// Mitsubishi GX Works2 project: compiler   PLC: FX3G

// global labels: Global1
VAR_GLOBAL
  AM_EVENTS : ARRAY [0..3] OF ST_AM_EVENT;
  AM_ALARMS : ARRAY [0..2] OF ST_AM_ALARM;
END_VAR
VAR_GLOBAL CONSTANT
  c_AM_ALARMS_NUM : INT := 3;
  c_AM_EVENTS_NUM : INT := 3;
END_VAR
VAR_GLOBAL
  MB_CHANNELS : ARRAY [0..2] OF ST_MB_REG_50;
END_VAR
VAR_GLOBAL CONSTANT
  c_MB_CHANNELS_NUM : INT := 2;
END_VAR

// task MAIN (event TRUE, interval 0, priority 31): MAIN
// task AM (event FALSE, interval T#100ms, priority 31): PRG_AM_TEST
// task TCO (event I750, interval 0, priority 26): PRG_TCO_TICKER_50
// task TCO_TEST (event FALSE, interval T#20ms, priority 31): PRG_TEST_TCO_50
// task MB (event FALSE, interval T#20ms, priority 31): PRG_MB_TEST
// user libraries (not included): AlarmManger, Modbus, TimeControl, UtilsV5

PROGRAM MAIN
VAR
  fbHyst : FB_HYST;  (* Heating regulator instance *)
  fbHystCool : FB_HYST_COOL;  (* Cooling regulator instance *)
  fbScaleAI : FB_SCALE_AI;  (* Host PLC analog input scaling instance *)
  fbL02ScaleAI : L02_SCALE_AI;  (* L02 module analog input scaling instance *)
  fbValve3P : FB_VALVE_3P;  (* 3-position valve control instance *)
  xSaveIp : BOOL;  (* Manual trigger: write IP settings (force TRUE) *)
  xValveEnable : BOOL;  (* Manual valve enable input *)
  xIsOnWord : BOOL;  (* F_ISBON result (bit 2 of 16#0004 = TRUE) *)
  xIsOnDword : BOOL;  (* F_DISBON result (bit 2 of 16#00000004 = TRUE) *)
  wSetWord : WORD;  (* F_SETB result (16#0000 with bit 3 set = 16#0008) *)
  dwSetWord : DWORD;  (* F_DSETB result (bit 3 set) *)
  wRstWord : WORD;  (* F_RSTB result (16#000F with bit 2 cleared = 16#000B) *)
  dwRstWord : DWORD;  (* F_DRSTB result (bit 2 cleared) *)
  wSrbWord : WORD;  (* F_SRB result (bit 5 set) *)
  dwSrbWord : DWORD;  (* F_DSRB result (bit 5 set) *)
  iLimit : INT;  (* F_LIMIT result (150 clamped to 100) *)
  iScale : INT;  (* F_SCALE result (50 -> 500) *)
  iScaleNl : INT;  (* F_SCALE_NL result *)
  iIncrement : INT;  (* F_INCN result (2 -> 3) *)
  iShift : INT;  (* F_SHFT result (4 shifted by 2 within 0..5 = 0) *)
  iWorkLeft : INT;  (* F_WORK_LEFT result (25/100 -> 75) *)
  iWorkLeftTime : INT;  (* F_WORK_LEFT_TIME result (25s/100s -> 75) *)
  iValvePos : INT;  (* F_VALVE_POS result (5s/10s -> 500) *)
  rFlt10 : REAL;  (* F_FLT10 result (123 -> 12.3) *)
  xSetIp : BOOL;  (* F_L02_SET_IP result *)
  xMbmov : BOOL;  (* F_MBMOV result *)
  xHystQ : BOOL;  (* FB_HYST output *)
  xHystCoolQ : BOOL;  (* FB_HYST_COOL output *)
  iScaleAIValue : INT;  (* FB_SCALE_AI scaled value *)
  xScaleAIWire : BOOL;  (* FB_SCALE_AI wire error *)
  xScaleAILimit : BOOL;  (* FB_SCALE_AI limit error *)
  xScaleAIMinMax : BOOL;  (* FB_SCALE_AI min/max error *)
  iL02ScaleAIValue : INT;  (* FB_L02_SCALE_AI scaled value *)
  xValveOpen : BOOL;  (* FB_VALVE_3P open command *)
  xValveClose : BOOL;  (* FB_VALVE_3P close command *)
END_VAR
EI(TRUE);

(*
  Utils library smoke test.

  Calls every function ( F_* ) and function block ( FB_* ) OF the Utils library
  with representative test inputs. Results are stored in auto-assigned labels
  so they can be watched in the device monitor.

  Functions exercised:
    F_ISBON / F_DISBON / F_SETB / F_DSETB / F_RSTB / F_DRSTB / F_SRB / F_DSRB
    F_LIMIT / F_SCALE / F_SCALE_NL / F_INCN / F_SHFT
    F_WORK_LEFT / F_WORK_LEFT_TIME / F_VALVE_POS / F_FLT10
    F_L02_SET_IP / F_MBMOV

  Function blocks exercised:
    FB_HYST / FB_HYST_COOL / FB_SCALE_AI / FB_L02_SCALE_AI / FB_VALVE_3P

  Notes:
    - FB_VALVE_3P uses the TCO_DINT_50 ticker AND therefore requires the
      TimeControl library with its TCO timer setup.
    - F_L02_SET_IP, F_MBMOV AND F_SCALE_NL write to R / D devices.
    - Force the xSaveIp / xValveEnable inputs AND watch the result labels.
*)

(* --- Bit check / bit manipulation functions --- *)
xIsOnWord  := F_ISBON(16#0004, 2);
xIsOnDword := F_DISBON(16#00000004, 2);

wSetWord  := F_SETB(16#0000, 3);
dwSetWord := F_DSETB(16#00000000, 3);

wRstWord  := F_RSTB(16#000F, 2);
dwRstWord := F_DRSTB(16#0000000F, 2);

wSrbWord  := F_SRB(16#0000, 5, TRUE);
dwSrbWord := F_DSRB(16#00000000, 5, TRUE);

(* --- Value / index functions --- *)
iLimit     := F_LIMIT(100, 150, 0);
iScale     := F_SCALE(50, 0, 100, 0, 1000);
iScaleNl   := F_SCALE_NL(2, 100, 50);  (* writes D100..D103 *)

iIncrement := F_INCN(TRUE, 2, 5);
iShift     := F_SHFT(2, 4, 5);

(* --- Progress / time functions --- *)
iWorkLeft     := F_WORK_LEFT(25, 100);
iWorkLeftTime := F_WORK_LEFT_TIME(T#25s, T#100s);
iValvePos     := F_VALVE_POS(T#5s, T#10s);

(* --- Filter function (returns REAL) --- *)
rFlt10 := F_FLT10(123);

(* --- Setup / command functions (device side effects) --- *)
(* Writes IP 192.168.0.100 to R23807/R23808 while xSaveIp is TRUE *)
xSetIp := L02_SET_IP(xSaveIp, IP_PLC_IP, 16#00C0, 16#00A8, 16#0000, 16#0064);

(* Copies 4 words D100..D103 to D200..D203 every scan *)
xMbmov := F_MBMOV(TRUE, 100, 4, 200);

(* --- Function blocks --- *)
(* Heating regulator: turns off when iPV < iSV *)
fbHyst(xIn := TRUE, iSV := 250, iPV := 200, iDV := 5, xQ := xHystQ);

(* Cooling regulator: turns off when iPV > iSV *)
fbHystCool(xIn := TRUE, iSV := 250, iPV := 200, iDV := 5, xQ := xHystCoolQ);

(* Analog input scaling (host PLC, D8030 area) *)
fbScaleAI(iAINum := 0, iSType := STYPE_4_20MA, iMin := 0, iMax := 160,
    iFilterTime := 10, iFilterNum := 100, iCorrection := 0,
    iValueOut := iScaleAIValue, xErrWire := xScaleAIWire,
    xErrLimit := xScaleAILimit, xErrMinMax := xScaleAIMinMax);

(* Analog input scaling (L02 modules, R23700 area) *)
fbL02ScaleAI(iAINum := 0, iSType := STYPE_4_20MA, iMin := 0, iMax := 160,
    iCorrection := 0, iValueOut := iL02ScaleAIValue);

(* 3-position valve control with position feedback *)
fbValve3P(xEnable := xValveEnable, iSV := 500, iDlt := 20,
    tTotalTime := T#10s, tLuftTime := T#500ms,
    xCloseOnDisable := TRUE, xIsOpened := FALSE, xIsClosed := FALSE,
    xOpen := xValveOpen, xClose := xValveClose);
END_PROGRAM
